TYPE ST_Kistler_CMD :
STRUCT

		bEnable		: BOOL;
		bAbort 		: BOOL;
		bStart		: BOOL;
		bReset		: BOOL;
		bManualMode	: BOOL;

END_STRUCT
END_TYPE

(* stored: Version 1.1.0.1
   DUT ST_Kistler_CMD: Id {5d01b955-fdcf-413e-a192-56838b56a525} *)
